/// enumeration of all possible priority
TYPE E_FilterActive :
(
	eFilter_none := 0,
	eFilter_activ := 1
);
END_TYPE

(* stored: Version 1.1.0.1
   DUT E_FilterActive: Id {7b98fbf7-ef6c-40b0-a4f2-4d05e82d2059} *)
